INTERFACE I_RpcInvoke

METHOD Invoke : ST_AdsStatus
VAR_INPUT
END_VAR
END_METHOD

END_INTERFACE

(* stored: Version 1.1.0.1, ProductVersion 3.1.4024.12
   Itf I_RpcInvoke: Id {c25a107c-452a-4c37-94bc-4b2d6880066d}
   Method Invoke: Id {d352277c-54f8-443f-a049-1475878c0922} *)
